KUKA KRL data list: RoboSyncControl.dat

&ACCESS RVO3
&REL 16
&PARAM DISKPATH = KRC:\R1\TP\CNCRobotics\CEAD
DEFDAT  RoboSyncControl PUBLIC
;************************************************
;     NextState Automation Ltd
;     www.nextstateautomation.co.uk
;************************************************
;     Contact: helpdesk@nextstate.co.uk
;     Date: 14/09/26
;     Version: 0.1.1
;************************************************

GLOBAL ENUM ENUM_PID_TYPE HEATED_BED, EXTRUDER0, EXTRUDER1, NOZZLE

GLOBAL CONST INT RESET_ALARM_CODE=186
GLOBAL CONST INT ENABLE_DRIVE=159
GLOBAL CONST INT DISABLE_DRIVE=158
GLOBAL CONST INT COMMENCE_JOGGING=150
GLOBAL CONST INT STOP_JOGGING=216
GLOBAL CONST INT MOVE_RELATIVE_DISTANCE=102
GLOBAL CONST INT MOVE_ABSOLUTE_DISTANCE=103
GLOBAL CONST INT FAST_STOP_MOVE=225
GLOBAL CONST INT STOP_MOVE=226
GLOBAL CONST INT SET_POSITION = 165

GLOBAL CONST INT AUTOTUNE_FAST=1
GLOBAL CONST INT AUTOTUNE_FULL=2
GLOBAL CONST INT AUTOTUNE_STOP=0

GLOBAL REAL pidDefaultUpperLimit=1.25
GLOBAL REAL pidDefaultLowerLimit=0.75


GLOBAL ENUM ENUM_STEPPER_PARAM CURRENT,IDLE_CURRENT,PULSE_PER_REV,JOG_SPEED,JOG_ACCEL,JOG_DECEL,SPEED,ACCEL,DECEL,DISTANCE,SET_POSITION


GLOBAL REAL rTemperatureTolerance = 10

GLOBAL CONST INT AUTOTUNE_TIMER=19
GLOBAL INT nAutotuneStartTimeout = 5000

ENDDAT
